// TwinCAT 3 PLC project plc_kfe_vac_fs
// ProgramVersion: 3.1.4023.0
// libraries:
//   LCLS General, * (SLAC)
//   LCLS Vacuum, * (SLAC - LCLS)
//   PMPS, * (SLAC - LCLS)
//   Tc2_Standard, * (Beckhoff Automation GmbH)
//   Tc2_System, * (Beckhoff Automation GmbH)
//   Tc3_Module, * (Beckhoff Automation GmbH)
// project tree:
//   GVLs/ GVL_SXR_VAC_FSV_PMPS.TcGVL, GVL_SXR_VAC_FS_DEVICES.TcGVL
//   / PlcTask.TcTTO
//   POUs/ MAIN.TcPOU
// (motion and I/O tree: see PLC project plc_kfe_vac)
// real-time tasks:
//   TASK PlcTask: cycle T#10ms, priority 20, ADS port 350
//   TASK SimTask: cycle T#10ms, priority 21, ADS port 351
//   TASK PlcTask1: cycle T#10ms, priority 22, ADS port 352
// variable links:
//   plc_kfe_vac_fs/plc_kfe_vac_fs Instance <-> Device 1 (EtherCAT)/=+-EK1100_02_00/=+-EL1124_02_08
//     PlcTask Inputs/GVL_SXR_VAC_FS_DEVICES.fb_TV2K0_VFS_1.i_xTrigger <-> Channel 1/GVL_SXR_VAC_FS_DEVICES.fb_TV2K0_VFS_1.i_xTrigger
//   plc_kfe_vac_fs/plc_kfe_vac_fs Instance <-> Device 1 (EtherCAT)/=+-EK1100_05_01/=+-ES1004_05_02
//     PlcTask Inputs/GVL_SXR_VAC_FS_DEVICES.fb_TV2K0_VFS_1.i_xClsLS <-> Channel 1/GVL_SXR_VAC_FS_DEVICES.fb_TV2K0_VFS_1.i_xClsLS
//     PlcTask Inputs/GVL_SXR_VAC_FS_DEVICES.fb_TV2K0_VFS_1.i_xOpnLS <-> Channel 2/GVL_SXR_VAC_FS_DEVICES.fb_TV2K0_VFS_1.i_xOpnLS
//   plc_kfe_vac_fs/plc_kfe_vac_fs Instance <-> Device 1 (EtherCAT)/=+-EK1100_05_01/=+-ES2202_05_03
//     PlcTask Outputs/GVL_SXR_VAC_FS_DEVICES.fb_TV2K0_VFS_1.q_xClose_A <-> Channel 1/GVL_SXR_VAC_FS_DEVICES.fb_TV2K0_VFS_1.q_xClose_A
//     PlcTask Outputs/GVL_SXR_VAC_FS_DEVICES.fb_TV2K0_VFS_1.q_xClose_B <-> Channel 2/GVL_SXR_VAC_FS_DEVICES.fb_TV2K0_VFS_1.q_xClose_B
//   plc_kfe_vac_fs/plc_kfe_vac_fs Instance <-> Device 1 (EtherCAT)/=+-EK1100_05_01/=+-ES2202_05_04
//     PlcTask Outputs/GVL_SXR_VAC_FS_DEVICES.fb_TV2K0_VFS_1.q_xClose_C <-> Channel 1/GVL_SXR_VAC_FS_DEVICES.fb_TV2K0_VFS_1.q_xClose_C
//     PlcTask Outputs/GVL_SXR_VAC_FS_DEVICES.fb_TV2K0_VFS_1.q_xOPN_DO <-> Channel 2/GVL_SXR_VAC_FS_DEVICES.fb_TV2K0_VFS_1.q_xOPN_DO

CONFIGURATION plc_kfe_vac_fs
    RESOURCE PLC ON TwinCAT3
        TASK PlcTask(INTERVAL := T#1ms, PRIORITY := 13);
        PROGRAM MAIN WITH PlcTask : MAIN;
    END_RESOURCE
END_CONFIGURATION

// ---- GVLs/GVL_SXR_VAC_FSV_PMPS.TcGVL
VAR_GLOBAL
    {attribute 'pytmc' := '
    	pv: PLC:KFE:VAC:K0:FF2
    '}
    {attribute 'TcLinkTo' := '.q_xFastFaultOut:=TIIB[PMPS_FFO (EL2202)]^Channel 2^Output'}
    g_FastFaultOutput2  :	FB_HardwareFFOutput;	//FFO for Fast Shutter Valves upstream of ST1L0_XTES
END_VAR

// ---- GVLs/GVL_SXR_VAC_FS_DEVICES.TcGVL
VAR_GLOBAL
	
    {attribute 'pytmc' := '
		pv: TV2K0:VFS:1
	'}
	fb_TV2K0_VFS_1 : FB_VFS;
END_VAR

// ---- POUs/MAIN.TcPOU
PROGRAM MAIN
VAR
END_VAR

fb_TV2K0_VFS_1(
	i_xPMPS_OK:= TRUE, 
	i_xExt_OK:= TRUE, 
	i_sDevName:= 'TV2K0:VFS:1',
	io_fbFFHWO:= g_FastFaultOutput2
);

(*FastFaultOuput*)	
g_FastFaultOutput2.Execute(bAutoReset:= TRUE);

END_PROGRAM
